FUNCTION_BLOCK FB_MZHeaterRef
VAR_INPUT
END_VAR
VAR_OUTPUT
	pMultiZRef 		: POINTER TO FB_MultiZRef;
	nChannel 		: USINT;
	nTemp1Actual 	AT %I* : UINT;
	nTemp2Actual 	AT %I* : UINT;
	nTemp3Actual 	AT %I* : UINT;	
	bHeaterIsOn		AT %I* : BOOL;
END_VAR
VAR
	bHeaterExistDetected	: BOOL;
	bHeaterExistFixed		: BOOL;
	nTemp1Setpoint	: UINT;
END_VAR

METHOD FB_init : BOOL
VAR_INPUT
	bInitRetains : BOOL; // if TRUE, the retain variables are initialized (warm start / cold start)
	bInCopyCode : BOOL;  // if TRUE, the instance afterwards gets moved into the copy code (online change)
	pMultiZRef 		: POINTER TO FB_MultiZRef;
END_VAR

VAR
	nFirstAdress : PVOID;
	nSelfAdress : PVOID;
END_VAR
THIS^.pMultiZRef := pMultiZRef;
nFirstAdress := ADR(pMultiZRef^.aFbHeaterRef);
nSelfAdress := THIS;
{IF hasvalue (RegisterSize, '32')}
nChannel := UDINT_TO_USINT((nSelfAdress - nFirstAdress)/SIZEOF(THIS^) + 1);
{ELSE}
nChannel := ULINT_TO_USINT((nSelfAdress - nFirstAdress)/SIZEOF(THIS^) + 1);
{END_IF}
END_METHOD

PROPERTY P_bHeaterDetected : BOOL
GET
P_bHeaterDetected := bHeaterExistDetected;
END_GET
SET
bHeaterExistDetected := P_bHeaterDetected;
END_SET
END_PROPERTY

PROPERTY P_bHeaterFixed : BOOL
GET
P_bHeaterFixed := bHeaterExistFixed;
END_GET
SET
bHeaterExistFixed := P_bHeaterFixed;
END_SET
END_PROPERTY

PROPERTY P_nTemp1Setpoint : UINT
GET
P_nTemp1Setpoint := nTemp1Setpoint;
END_GET
SET
nTemp1Setpoint := P_nTemp1Setpoint;
END_SET
END_PROPERTY

END_FUNCTION_BLOCK

(* stored: Version 1.1.0.1, ProductVersion 3.1.4022.18
   POU FB_MZHeaterRef: Id {65c87e2f-4183-4293-8be1-f16cff76eb5a}, SpecialFunc None
   Method FB_init: Id {d3e74796-9cf6-4ba6-9718-4727b951d51e}
   Property P_bHeaterDetected: Id {12c075e0-4a35-4347-b611-72372288168c}
   Get Get: Id {77f28342-85fe-441f-9fba-41470b6cbe76}
   Set Set: Id {18556449-fe3f-47af-8ab3-e3d571e72d8e}
   Property P_bHeaterFixed: Id {9fbe1f83-07bb-4738-8b99-3eddcc55f066}
   Get Get: Id {a31725dd-d735-477e-9ad2-16243126793e}
   Set Set: Id {037c7b4d-a7c3-42d9-a593-cf990456ca32}
   Property P_nTemp1Setpoint: Id {baa31b71-6661-46a3-82e0-1f1b8b7622ed}
   Get Get: Id {2b2734ba-fb4d-4e93-a9aa-3cd275b4c657}
   Set Set: Id {cc6931de-5147-4618-abb4-130c709e723d} *)
